// TIA Portal V20 export
TYPE "UDT_Service_ServProcessParameter"
   STRUCT
      Analog : Array[0..31] of "UDT_MTP_AnaProcessValueIn";
      Digital : Array[0..7] of "UDT_MTP_DIntProcessValueIn";
      Binary : Array[0..31] of "UDT_MTP_BinProcessValueIn";
      "String" : Array[0..7] of "UDT_MTP_StringProcessValueIn";
   END_STRUCT;
END_TYPE
